// TwinCAT 3 PLC project PLC
// ProgramVersion: 3.1.4023.0
// libraries:
//   Tc2_Standard, * (Beckhoff Automation GmbH)
//   Tc2_System, * (Beckhoff Automation GmbH)
//   Tc3_Module, * (Beckhoff Automation GmbH)
// project tree:
//   / PlcTask.TcTTO
//   POUs/ ACMotor.TcPOU, ContactorNO.TcPOU, LedLamp.TcPOU, MAIN.TcPOU, SignalTower.TcPOU
//   POUs/Buttons/ Button.TcPOU, ButtonNO.TcPOU, ButtonNC.TcPOU
// real-time tasks:
//   TASK PlcTask: cycle T#10ms, priority 20, ADS port 350

CONFIGURATION PLC
    RESOURCE PLC ON TwinCAT3
        TASK PlcTask(INTERVAL := T#10ms, PRIORITY := 20);
        PROGRAM MAIN WITH PlcTask : MAIN;
    END_RESOURCE
END_CONFIGURATION

// ---- POUs/MAIN.TcPOU
PROGRAM MAIN
VAR
	motor	 			: ACMotor;
	motorChangeTimer 	: TON;
	
	startButton			: ButtonNO;
	signalTower			: SignalTower;
END_VAR

MotionLogic();
SignalTowerLogic();

METHOD MotionLogic
IF startButton.IsPressed THEN
	motorChangeTimer(
		IN := NOT motorChangeTimer.Q,
		PT := T#10S);
	
	IF motorChangeTimer.Q AND_THEN motor.IsMoving THEN
		motor.Stop();
	ELSIF motorChangeTimer.Q THEN
		motor.Start();
	END_IF
ELSE
	motorChangeTimer(IN := FALSE);
	motor.Stop();
END_IF
END_METHOD

METHOD SignalTowerLogic
VAR_INPUT
END_VAR
IF startButton.IsPressed THEN
	signalTower.SetStateOP();
ELSE
	signalTower.SetStateSTOP();
END_IF
END_METHOD

END_PROGRAM

// ---- POUs/ACMotor.TcPOU
FUNCTION_BLOCK ACMotor
VAR
	moveContactor : ContactorNO;
END_VAR

PROPERTY IsMoving : BOOL
GET
IsMoving := moveContactor.IsClosed;
END_GET
END_PROPERTY

METHOD Start
VAR_INPUT
END_VAR
moveContactor.Close();
END_METHOD

METHOD Stop
VAR_INPUT
END_VAR
moveContactor.Open();
END_METHOD

END_FUNCTION_BLOCK

// ---- POUs/ContactorNO.TcPOU
FUNCTION_BLOCK ContactorNO
VAR
	output AT %Q* : BOOL;
END_VAR

METHOD Close
VAR_INPUT
END_VAR
output := TRUE;
END_METHOD

PROPERTY IsClosed : BOOL
GET
IsClosed := output;
END_GET
END_PROPERTY

PROPERTY IsOpen : BOOL
GET
IsOpen := NOT output;
END_GET
END_PROPERTY

METHOD Open
VAR_INPUT
END_VAR
output := FALSE;
END_METHOD

END_FUNCTION_BLOCK

// ---- POUs/Buttons/ButtonNO.TcPOU
FUNCTION_BLOCK ButtonNO EXTENDS Button
VAR
	input AT %I* : BOOL;
END_VAR

PROPERTY IsPressed : BOOL
GET
IsPressed := input;
END_GET
END_PROPERTY

PROPERTY IsReleased : BOOL
GET
IsReleased := NOT input;
END_GET
END_PROPERTY

END_FUNCTION_BLOCK

// ---- POUs/Buttons/Button.TcPOU
FUNCTION_BLOCK ABSTRACT Button
VAR
	input AT %I* : BOOL;
END_VAR

PROPERTY PUBLIC State : BOOL
GET
state := input;
END_GET
END_PROPERTY

END_FUNCTION_BLOCK

// ---- POUs/SignalTower.TcPOU
FUNCTION_BLOCK SignalTower
VAR
	ledRed		: LedLamp;
	ledGreen	: LedLamp;
END_VAR

METHOD SetStateOP
VAR_INPUT
END_VAR
ledRed.Off();
ledGreen.On();
END_METHOD

METHOD SetStateSTOP
VAR_INPUT
END_VAR
ledRed.On();
ledGreen.Off();
END_METHOD

END_FUNCTION_BLOCK

// ---- POUs/LedLamp.TcPOU
FUNCTION_BLOCK LedLamp
VAR_INPUT
END_VAR
VAR_OUTPUT
END_VAR
VAR
	output AT %Q* : BOOL;
END_VAR

PROPERTY IsOff : BOOL
GET
IsOff := NOT output;
END_GET
END_PROPERTY

PROPERTY IsOn : BOOL
GET
IsOn := output;
END_GET
END_PROPERTY

METHOD Off
VAR_INPUT
END_VAR
output := FALSE;
END_METHOD

METHOD On
VAR_INPUT
END_VAR
output := TRUE;
END_METHOD

END_FUNCTION_BLOCK

// ---- POUs/Buttons/ButtonNC.TcPOU
FUNCTION_BLOCK ButtonNC EXTENDS Button
VAR
	input AT %I* : BOOL;
END_VAR

PROPERTY IsPressed : BOOL
GET
IsPressed := NOT input;
END_GET
END_PROPERTY

PROPERTY IsReleased : BOOL
GET
IsReleased := input;
END_GET
END_PROPERTY

END_FUNCTION_BLOCK
